FUNCTION_BLOCK Control
VAR_INPUT
END_VAR
VAR_OUTPUT
END_VAR
VAR
END_VAR

END_FUNCTION_BLOCK

(* stored: Version 1.1.0.1, ProductVersion 3.1.4024.0
   POU Control: Id {4ac48026-8297-495a-80fd-a44f599bcfa3}, SpecialFunc None *)
